PROGRAM pouStationLangauge
VAR
	row1: FB_HMI_Control;
	row2: FB_HMI_Control;
	row3: FB_HMI_Control;
	row4: FB_HMI_Control;
	row5: FB_HMI_Control;
	row6: FB_HMI_Control;
	row7: FB_HMI_Control;
	row8: FB_HMI_Control;
	row9: FB_HMI_Control;
	row10: FB_HMI_Control;
	tNumberOfPages: REAL;
	tCalcNumberOfPages: REAL;
	row11: FB_HMI_Control;
	row12: FB_HMI_Control;
	row13: FB_HMI_Control;
	row14: FB_HMI_Control;
	row15: FB_HMI_Control;
	row16: FB_HMI_Control;
	row17: FB_HMI_Control;
	row18: FB_HMI_Control;
	row19: FB_HMI_Control;
	row20: FB_HMI_Control;
	row21: FB_HMI_Control;
	row22: FB_HMI_Control;
	row23: FB_HMI_Control;
	row24: FB_HMI_Control;
	//StationNativeMotionRows: ARRAY[0..99] OF typeMotionRow;
	ceil: LREAL;
END_VAR

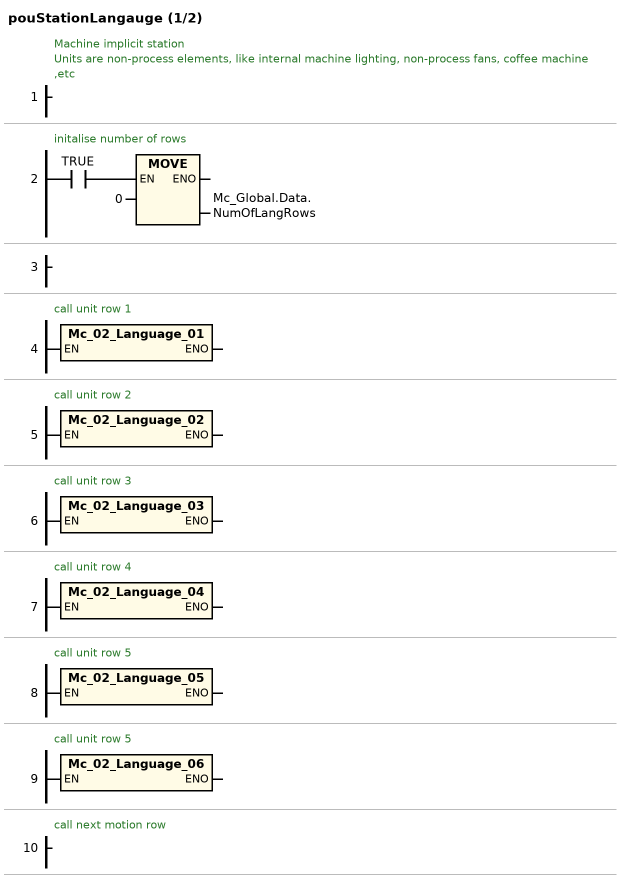
// NETWORK 1
// Machine implicit station
// Units are non-process elements, like internal machine lighting, non-process fans, coffee machine ,etc

// NETWORK 2
// initalise number of rows
Mc_Global.Data.NumOfLangRows := 0;

// NETWORK 3

// NETWORK 4
// call unit row 1
Mc_02_Language_01();

// NETWORK 5
// call unit row 2
Mc_02_Language_02();

// NETWORK 6
// call unit row 3
Mc_02_Language_03();

// NETWORK 7
// call unit row 4
Mc_02_Language_04();

// NETWORK 8
// call unit row 5
Mc_02_Language_05();

// NETWORK 9
// call unit row 5
Mc_02_Language_06();

// NETWORK 10
// call next motion row

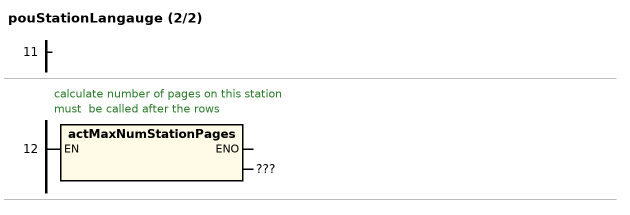
// NETWORK 11

// NETWORK 12
// calculate number of pages on this station
// must  be called after the rows
actMaxNumStationPages();

ACTION actMaxNumStationPages:
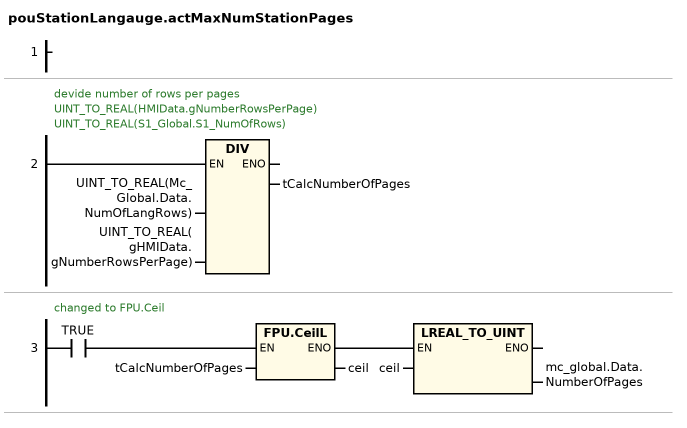
// NETWORK 1

// NETWORK 2
// devide number of rows per pages
// UINT_TO_REAL(HMIData.gNumberRowsPerPage)
// UINT_TO_REAL(S1_Global.S1_NumOfRows)
tCalcNumberOfPages := (UINT_TO_REAL(Mc_Global.Data.NumOfLangRows)) / (UINT_TO_REAL(gHMIData.gNumberRowsPerPage));

// NETWORK 3
// changed to FPU.Ceil
ceil := FPU.CeilL(tCalcNumberOfPages);
mc_global.Data.NumberOfPages := LREAL_TO_UINT(ceil);
END_ACTION

END_PROGRAM

(* stored: Version 1.1.0.1, ProductVersion 3.1.4024.12
   POU pouStationLangauge: Id {714f5004-1402-4d18-9e82-2807c38c6337}, SpecialFunc None
   Action actMaxNumStationPages: Id {9ab21fdf-75fa-4a93-808b-5169061f4680} *)
